// Mitsubishi GX Works2 project: 0710-incZ1   PLC: Q02/Q02H

PROGRAM MAIN
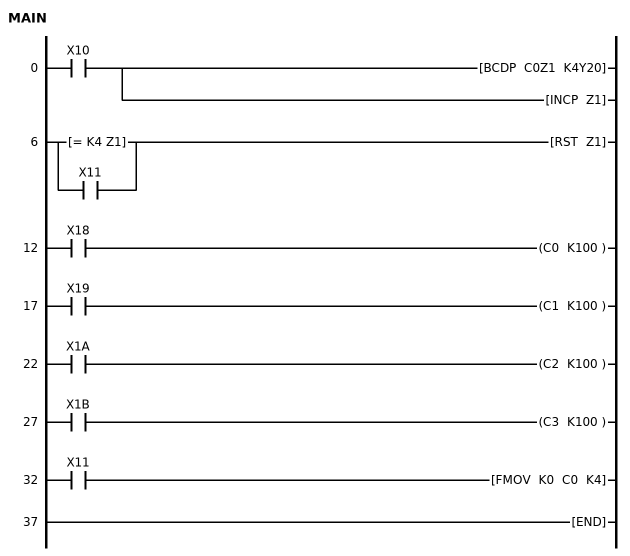
0     LD      X10
      BCDP    C0Z1 K4Y20
      INCP    Z1
6     LD=     K4 Z1
      OR      X11
      RST     Z1
12    LD      X18
      OUT     C0 K100
17    LD      X19
      OUT     C1 K100
22    LD      X1A
      OUT     C2 K100
27    LD      X1B
      OUT     C3 K100
32    LD      X11
      FMOV    K0 C0 K4
37    END
END_PROGRAM
